FUNCTION_BLOCK Git_Test
VAR_INPUT
END_VAR
VAR_OUTPUT
END_VAR
VAR
END_VAR

Hallo Jan ausm GIT

END_FUNCTION_BLOCK

(* stored: Version 1.1.0.1, ProductVersion 3.1.4026.11
   POU Git_Test: Id {9f67af42-6a8e-4204-8caf-9413ae67d438}, SpecialFunc None *)
